TYPE T_Hashmap_Bucket_Node : ST_HASHMAP_BUCKET_NODE; END_TYPE

(* stored: Version 1.1.0.1
   DUT T_Hashmap_Bucket_Node: Id {75699d58-a158-0d87-3e7a-7773b888a364} *)
